(* PLC project Command Pattern Example.project, CODESYS CODESYS V3.5 SP20 Patch 1 *)
(* stored: creationDateTime 2025-05-27T21:23:14.9949448, modificationDateTime 2025-05-27T21:22:47.7198131 *)

INTERFACE ICommand
METHOD Execute
END_METHOD
END_INTERFACE

PROGRAM PLC_PRG
  VAR
    Commands : CommandQueue;
    currentCommand : ICommand;
    canExecute : BOOL;
    isDequeued : BOOL;
    startPump : PurgeCommand;  (* Command objects *)
    stopPump : CleanCommand;
  END_VAR

                    
IF Commands.IsCommandPending  AND canExecute THEN
	isDequeued := Commands.Dequeue(ADR(currentCommand));
END_IF
	
IF isDequeued THEN
	currentCommand.Execute();
	isDequeued := FALSE;
END_IF


                  
END_PROGRAM

FUNCTION_BLOCK CommandQueue
  VAR CONSTANT
    MaxSize : BYTE := 10;
  END_VAR
  VAR
    _head : BYTE;
    _tail : BYTE;
    _count : BYTE;
    _commandBuffer : ARRAY[0..(MaxSize - 1)] OF ICommand;
  END_VAR

                    

                  

METHOD Dequeue : BOOL
  VAR_INPUT
    command : POINTER TO ICommand;
  END_VAR
                          
IF _count > 0 AND command > 0 THEN
    command^ := _commandBuffer[_head];
	_head := (_head + 1) MOD MaxSize;
    _count := _count - 1;
	
	Dequeue := TRUE;
ELSE
	Dequeue := FALSE;
END_IF
                        
END_METHOD

METHOD Enqueue : BOOL
  VAR_INPUT
    command : ICommand;
  END_VAR
                          
IF _count < MaxSize THEN
    _commandBuffer[_tail] := command;
    _tail := (_tail + 1) MOD MaxSize;
    _count := _count + 1;
	
    Enqueue := TRUE;
ELSE
    Enqueue := FALSE;
END_IF


                        
END_METHOD

PROPERTY IsCommandPending : BOOL
GET
                            
IsCommandPending := _count > 0;
                          
END_GET
END_PROPERTY
END_FUNCTION_BLOCK

FUNCTION_BLOCK MachineControl

                    
                  

METHOD Run : BOOL
                          
                        
END_METHOD

METHOD Stop : BOOL
                          
                        
END_METHOD

METHOD Clean : BOOL
                          
                        
END_METHOD

METHOD Purge : BOOL
                          
                        
END_METHOD
END_FUNCTION_BLOCK

FUNCTION_BLOCK PurgeCommand IMPLEMENTS ICommand
  VAR_IN_OUT
    Machine : MachineControl;
  END_VAR

                    
                  

METHOD Execute
                          
// Perform some checks
Machine.Run();
                        
END_METHOD
END_FUNCTION_BLOCK

FUNCTION_BLOCK CleanCommand IMPLEMENTS ICommand
  VAR_IN_OUT
    Machine : MachineControl;
  END_VAR

                    
                  

METHOD Execute
                          
// Perform some pre-checks
Machine.Clean();
                        
END_METHOD
END_FUNCTION_BLOCK

CONFIGURATION Device
  RESOURCE Application ON PLC
    TASK MainTask(INTERVAL := T#20ms, PRIORITY := 1);
    PROGRAM PLC_PRG WITH MainTask : PLC_PRG;
  END_RESOURCE
END_CONFIGURATION
